FUNCTION_BLOCK EL3443
VAR
	_io : EL3443_Data;
	{attribute addProperty Name "WcState"}
	_wcState : WcStateInputToggle;
	{attribute addProperty Name "Info data"}
	_infoData : InfoDataAds;
END_VAR

PROPERTY IO : REFERENCE TO EL3443_Data
GET
IO REF= _io;
END_GET
END_PROPERTY

PROPERTY WcState : REFERENCE TO WcStateInputToggle
GET
WcState REF= _wcState;
END_GET
END_PROPERTY

END_FUNCTION_BLOCK

(* stored: Version 1.1.0.1, ProductVersion 3.1.4024.9
   POU EL3443: Id {f2a4328a-b8aa-03e2-2bd5-fd6bfd729fab}, SpecialFunc None
   Property IO: Id {cfaa088a-517d-0d38-3b68-2a415355f805}
   Get Get: Id {5de58be2-51ff-077b-1c84-28cc5563f74a}
   Property WcState: Id {e8a672a3-df13-08b5-136b-e11edda6362d}
   Get Get: Id {5e49a863-63a9-0dd6-2148-957edbe25580} *)
